{attribute 'qualified_only'}
VAR_GLOBAL
	bSetNewMaxFlowCapacity		: BOOL;
	fNewMaxFlowCapacity 		: LREAL;
	bSetNewProportionalGain 	: BOOL;
	bSetNewIntegralGain 		: BOOL;
	fNewProportionalGain 		: LREAL;
	fNewIntegralGain 			: LREAL;
	bSetNewMaxPositionError 			: BOOL;
	fNewMaxPositionError				: LREAL;
	stAutomaticControlSettings 	: ST_AutomaticControlSettings;
	stMotionReferenceGeneratorSettings  : ST_MotionReferenceGeneratorSettings;
	SetPointVar : LREAL;
END_VAR

(* stored: Version 1.1.0.1, ProductVersion 3.1.4024.12
   GVL G_Commissioning: Id {f52cce8a-bb8c-4e23-918d-1587f9fb00ff} *)
